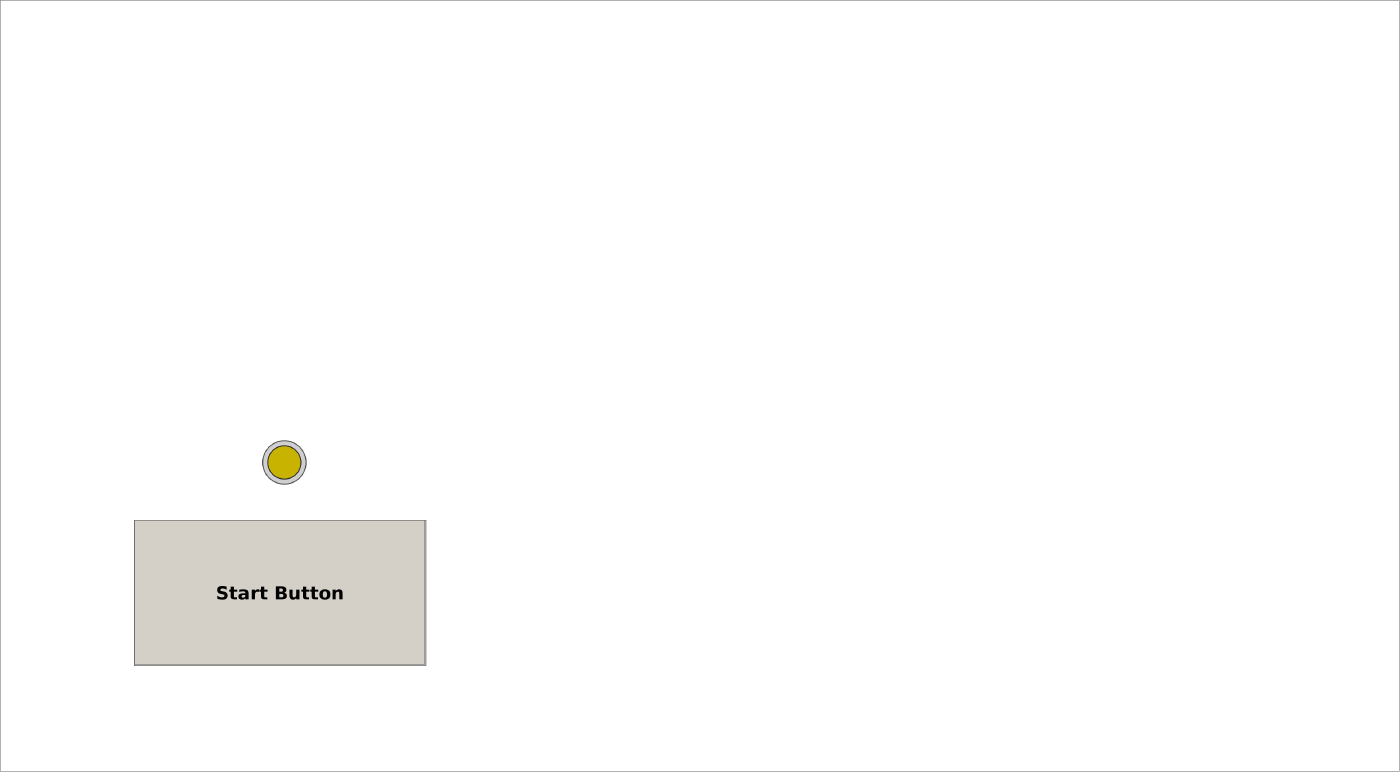
VISUALIZATION HOME_PAGE  // 1920x1060, background image ImagePool.Grey_Gradient
    Button (184,714 400x200), "Start Button"
        toggle OP_BTN.Start_btn
    Lamp1 (355,600 70x70), variable: OP_BTN.Start_lamp, style: Lamp-Lamp1-Yellow
END_VISUALIZATION

(* stored: Version 1.1.0.1, ProductVersion 3.1.4024.12
   Visu HOME_PAGE: Id {d910f869-af87-4472-b9bf-bcfb1b401c7c} *)
